TYPE ST_LSPM_Outp_Lift :
STRUCT
	LiftUp				: BOOL; //Move lift up
	LiftDown			: BOOL; //Move lift down
	LiftCS				: BOOL; // Move lift in creep speed	
END_STRUCT
END_TYPE

(* stored: Version 1.1.0.1, ProductVersion 3.1.4024.4
   DUT ST_LSPM_Outp_Lift: Id {24f1510a-b422-4ff6-a89e-e947a9ab5242} *)
